FUNCTION LogString : BOOL
VAR_INPUT
	sString: T_MaxString;
END_VAR

ADSLOGSTR(
	msgCtrlMask := ADSLOG_MSGTYPE_HINT,
	msgFmtStr := '%s',
	strArg := sString
);

END_FUNCTION

(* stored: Version 1.1.0.1, ProductVersion 3.1.4024.3
   POU LogString: Id {f5b2e333-f0e5-4c09-b1d1-9c9fa6989ae9}, SpecialFunc None *)
